RoboDK station: assembly_zone.rdk

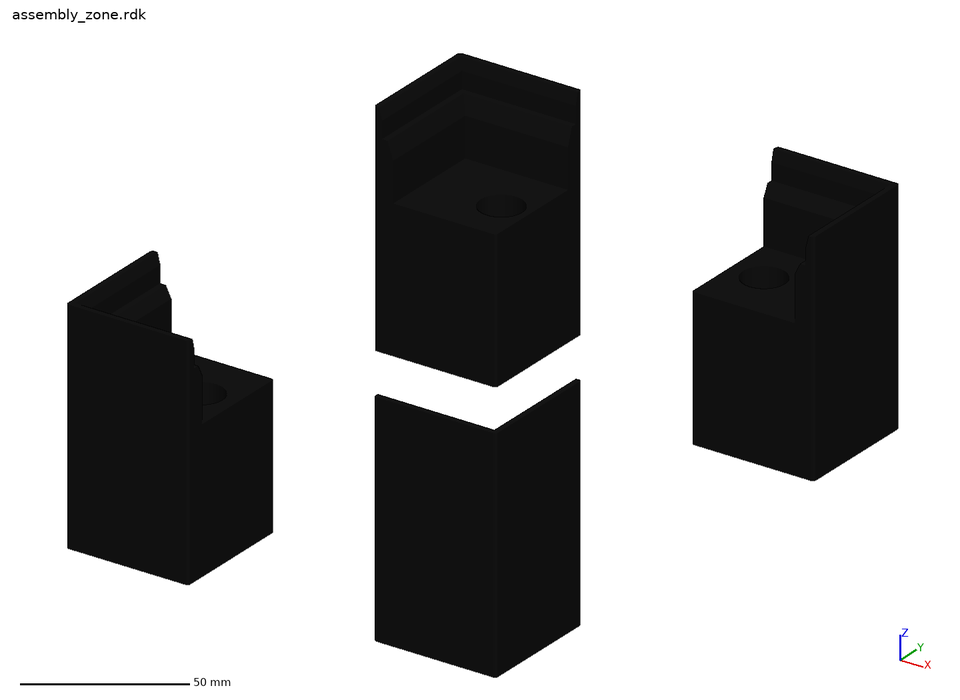
[picture v0: the station drawn from its stored meshes, robots at their saved joint values, targets as dots, program paths as lines]
Station assembly_station (saved by RoboDK 5.9.0). Poses are relative to the parent item; angles as X-Y-Z fixed-axis rotations.
  - object assembly_station at (0, 0, 0) mm, size 157 x 207 x 80 mm, geometry from assembly_station.stl
